// TIA Portal project "WEB" (V14)

(* hardware
DEVICE "S7-1200 station_1"  S7-1200 Station
   slot 0: "Rack_0"  S7-1200 Rack  Rack  V1.0
   slot 1: "PLC_1"  CPU 1214C DC/DC/DC  6ES7 214-1AG31-0XB0  V3.0
*)

// ===== PLC "PLC_1"  CPU 1214C DC/DC/DC =====

VAR_GLOBAL   // PLC tag table "Default tag table"
   "Motor" AT %Q0.0 : Bool;
   "Tag_2" AT %Q0.1 : Bool;
   "Start" AT %M0.0 : Bool;
   "Stop" AT %M0.1 : Bool;
   "Lỗi" AT %MW2 : Int;
   "Tag_1" AT %M2.0 : Bool;
   "System_Byte" AT %MB1 : Byte;
   "FirstScan" AT %M1.0 : Bool;
   "DiagStatusUpdate" AT %M1.1 : Bool;
   "AlwaysTRUE" AT %M1.2 : Bool;
   "AlwaysFALSE" AT %M1.3 : Bool;
   "Clock_Byte" AT %MB5 : Byte;
   "Clock_10Hz" AT %M5.0 : Bool;
   "Clock_5Hz" AT %M5.1 : Bool;
   "Clock_2.5Hz" AT %M5.2 : Bool;
   "Clock_2Hz" AT %M5.3 : Bool;
   "Clock_1.25Hz" AT %M5.4 : Bool;
   "Clock_1Hz" AT %M5.5 : Bool;
   "Clock_0.625Hz" AT %M5.6 : Bool;
   "Clock_0.5Hz" AT %M5.7 : Bool;
END_VAR

DATA_BLOCK "Data"   // DB1
{ S7_Optimized_Access := 'FALSE' }
VERSION : 0.1
   VAR
      Giatri : Word;
      "time" : Time;
      Start : Bool;
      Stop : Bool;
      Value : Array[0..10] of Word;
   END_VAR
BEGIN
END_DATA_BLOCK

// folder: System blocks/Program resources

DATA_BLOCK "IEC_Counter_0_DB"   // DB2
{ S7_Optimized_Access := 'TRUE' }
AUTHOR : Simatic
FAMILY : IEC
NAME : CNTR
VERSION : 1.0
// stored: InstanceOfName IEC_COUNTER
"IEC_COUNTER"
BEGIN
END_DATA_BLOCK

// folder: (top level)

ORGANIZATION_BLOCK "Main"   // OB1, LAD, ProgramCycle
TITLE = "Main Program Sweep (Cycle)"
{ S7_Optimized_Access := 'TRUE' }
VERSION : 0.1
BEGIN

REGION Network 1
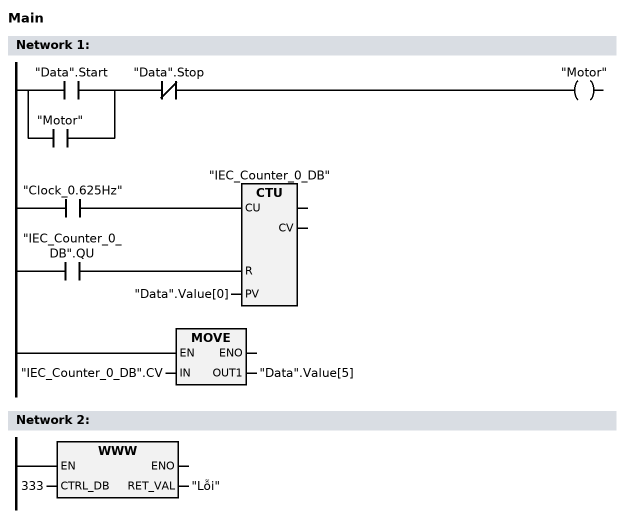
   "Motor" := ("Data".Start OR "Motor") AND NOT "Data".Stop;
   "IEC_Counter_0_DB".CTU(CU := "Clock_0.625Hz", R := "IEC_Counter_0_DB".QU, PV := "Data".Value[0]);
   "Data".Value[5] := "IEC_Counter_0_DB".CV;
END_REGION

REGION Network 2
   "Lỗi" := WWW(CTRL_DB := 333);
END_REGION
END_ORGANIZATION_BLOCK